SUBAPPLICATION Softkey_Aux_Method_Button_IE (* Softkey_Aux_Method_IE (SoftKey ODER AUX ODER lokale OPC-UA-Methode) ODER zusaetzlich ein weiterer Button (Button_IE, eigener CButton - z.B. IO-Diag-Testbutton, kann aber auch ein regulaerer Button sein) aktiviert -> 1 gemeinsames IND-Event. Fuer Ausgaenge, die sowohl echt bedient (SoftKey/AUX/Web/Dashboard) als auch per zusaetzlichem Button gleichberechtigt getriggert werden sollen - Background des Buttons wird vom Aufrufer separat aus dem resultierenden Zustand gespeist (dafuer bleibt u16ObjIdB beim Aufrufer verfuegbar). *)
  (* Standard: 61499-2; Description: Copyright (c) 2026 Meisterschulen am Ostbahnhof This program and the accompanying materials are made available under the terms of the Eclipse Public License 2.0 which is available at https://www.eclipse.org/legal/epl-2.0/ SPDX-License-Identifier: EPL-2.0 *)
  (* Version 1.1, 2026-09-15, Franz Höpfinger, Meisterschulen am Ostbahnhof, u16ObjId_TEST auf u16ObjIdB umbenannt (Button_IE_TEST -> Button_IE_B) - dieser zusaetzliche Button ist nicht immer nur ein IO-Diag-Testbutton, kann auch ein regulaerer Button sein. *)
  PACKAGE MyLib::sys;
  IMPORT isobus::UT::Q::const::IDs::ID_NULL;
  IMPORT isobus::UT::io::Button::ButtonActivationCode::BT_RELEASED_UNLATCHED;
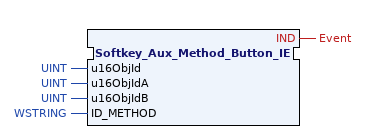
  EVENT_OUTPUT
    IND; (* Feuert wenn SoftKey, AUX, die lokale Methode ODER der IO-Diag-Testbutton aktiviert/aufgerufen wird *)
  END_EVENT
  VAR_INPUT
    u16ObjId : UINT; (* Object ID SoftKey *)
    u16ObjIdA : UINT; (* Object ID AuxFunction2 *)
    u16ObjIdB : UINT := ID_NULL; (* Object ID weiterer Button (z.B. IO-Diag-Testbutton, Ausgaenge-Diagnoseseite - kann aber auch ein regulaerer Button sein), gleichberechtigt zu SoftKey/AUX/Methode *)
    ID_METHOD : WSTRING; (* Lokale Methodenadresse (ACTION=CREATE_METHOD) fuer den argumentlosen Trigger - wird von Web-Client (vt-ui-mirror) UND direkt vom OPC-Dashboard aufgerufen *)
  END_VAR
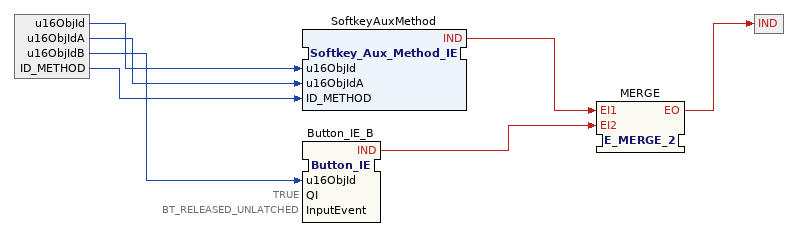
  FBS
    Button_IE_B : isobus::UT::io::Button::Button_IE(QI := TRUE, InputEvent := BT_RELEASED_UNLATCHED);
    MERGE : iec61499::events::E_MERGE_2;
  END_FBS
  SUBAPPS
    SoftkeyAuxMethod : MyLib::sys::Softkey_Aux_Method_IE;
  END_SUBAPPS
  EVENT_CONNECTIONS
    SoftkeyAuxMethod.IND TO MERGE.EI1;
    Button_IE_B.IND TO MERGE.EI2;
    MERGE.EO TO IND;
  END_CONNECTIONS
  DATA_CONNECTIONS
    u16ObjId TO SoftkeyAuxMethod.u16ObjId;
    u16ObjIdA TO SoftkeyAuxMethod.u16ObjIdA;
    ID_METHOD TO SoftkeyAuxMethod.ID_METHOD;
    u16ObjIdB TO Button_IE_B.u16ObjId;
  END_CONNECTIONS
END_SUBAPPLICATION
